PROGRAM MAIN
VAR
END_VAR

END_PROGRAM

(* stored: Version 1.1.0.1
   POU MAIN: Id {94ef9525-7cd5-4605-b8b6-a23a4b387845} *)
